// TwinCAT 3 PLC project nadaCAT
// ProgramVersion: 3.1.4024.0
// libraries:
//   Tc2_MC2, * (Beckhoff Automation GmbH)
//   Tc2_MC2_Drive, * (Beckhoff Automation GmbH)
//   Tc2_Standard, * (Beckhoff Automation GmbH)
//   Tc2_System, * (Beckhoff Automation GmbH)
//   Tc2_TcpIp, * (Beckhoff Automation GmbH)
//   Tc2_Utilities, * (Beckhoff Automation GmbH)
//   Tc3_Module, * (Beckhoff Automation GmbH)
//   VisuDialogs, * (System)
//   VisuSymbols,3.5.10.0,System
// project tree:
//   DUTs/Enums/ E_CommandList.TcTLEO (not stored), E_ServoState.TcTLEO, E_TCPState.TcTLEO (not stored)
//   DUTs/Structs/ dutCommand.TcDUT, mcInterface.TcDUT (not stored), mcOutputs.TcDUT (not stored), stConfigParams.TcDUT (not stored), stServoInterface.TcDUT (not stored), stStateTransitions.TcDUT
//   / GlobalTextList.TcGTLO (not stored), PlcTask.TcTTO (not stored), Visualization Manager.TcVMO (not stored), VISU_TASK.TcTTO
//   GVLs/ gvlMotion.TcGVL, IO.TcGVL, PLCSystem.TcGVL, ServoGVLs.TcGVL
//   POUs/FBs/ FB_AutoMotionControl.TcPOU (not stored), FB_ManualMotionControl.TcPOU, fb_StateMachine.TcPOU, FB_TCPServer.TcPOU, sfc_TCPServer.TcPOU
//   POUs/ MAIN.TcPOU
//   POUs/PRGs/ Motion.TcPOU (not stored), System.TcPOU (not stored), TCPComm.TcPOU
//   VISUs/ Main.TcVIS
//   VISUs/Templates/ MotorFaceplate.TcVIS, MotorFaceplate2.TcVIS, SysPanel.TcVIS

CONFIGURATION nadaCAT
    RESOURCE PLC ON TwinCAT3
        TASK VISU_TASK(INTERVAL := T#200000us, PRIORITY := 30);
        PROGRAM VisuElems_Visu_Prg WITH VISU_TASK : VisuElems.Visu_Prg;
    END_RESOURCE
END_CONFIGURATION

// ---- DUTs/Enums/E_ServoState.TcTLEO
{attribute 'qualified_only'}
{attribute 'strict'}
TYPE E_ServoState :
(
	DEFAULT	  := -1,
	OFF		  := 0,
	DISABLED,
	FAULTED,
	ENABLED,
	STANDBY,
	HOMING,
	MOVE_ABS,
	MOVE_REL,
	MOVE_SCAN,
	INTERLOCK_MOTION
);
END_TYPE
//  DEFAULT = '-1'

// ---- DUTs/Structs/dutCommand.TcDUT
TYPE dutCommand :
STRUCT
	eCommand 	: E_CommandList;
	arrParam	: ARRAY [1..5] OF LINT;
END_STRUCT
END_TYPE

// ---- DUTs/Structs/stStateTransitions.TcDUT
TYPE stStateTransitions :
STRUCT
	Init			: BOOL := FALSE;
	Standby			: BOOL := FALSE;
	cmdReceived		: BOOL := FALSE;
	cmdHome			: BOOL := FALSE;
	cmdScan			: BOOL := FALSE;
	cmdMTP			: BOOL := FALSE;
	cmdMovr			: BOOL := FALSE;
	cmdMova			: BOOL := FALSE;
	cmdStat			: BOOL := FALSE;
	cmdCal			: BOOL := FALSE;
	cmdParam		: BOOL := FALSE;
	cmdHomeDone		: BOOL := FALSE;
	cmdScanDone		: BOOL := FALSE;
	cmdMTPDone		: BOOL := FALSE;
	cmdMovrDone		: BOOL := FALSE;
	cmdMovaDone		: BOOL := FALSE;
	cmdStatDone		: BOOL := FALSE;
	cmdCalDone		: BOOL := FALSE;
	cmdParamDone	: BOOL := FALSE;
	cmdComplete		: BOOL := FALSE;
END_STRUCT
END_TYPE

// ---- GVLs/gvlMotion.TcGVL
{attribute 'qualified_only'}
VAR_GLOBAL
// Manual Control
servo1			: FB_ManualMotionControl;
bank1			: FB_AutoMotionControl;
manualMode 		: BOOL := TRUE;
autoMode		: BOOL;
// Server Control
cmdData 		: dutCommand;
bEnableDrive	: BOOL := FALSE;
bStartDrive		: BOOL := FALSE;
bTriggerDefault : BOOL := FALSE;
bInterlockOK	: BOOL := TRUE;
mcBankAxis		: stServoInterface;
driveStatus 	: ST_AxisStatus;	
END_VAR

// ---- GVLs/IO.TcGVL
{attribute 'qualified_only'}
VAR_GLOBAL
	/// Inputs
	bHomeSwitch 		AT %I* : BOOL;
	/// Outputs
	
END_VAR

// ---- GVLs/PLCSystem.TcGVL
{attribute 'qualified_only'}
VAR_GLOBAL
	iTaskIdx 	: DINT;
	bFirstCycle : BOOL;
END_VAR

// ---- GVLs/ServoGVLs.TcGVL
{attribute 'qualified_only'}
VAR_GLOBAL
	servo1Interface		: stServoInterface;
	servo2Interface		: stServoInterface;
	
	rTorqueLimit AT %Q*		: INT;
	rTorqueAct	 AT %I*		: INT;
	
	probe1Signal AT %I*		: WORD;
	probe1NegLatch AT %I*		: WORD;
	probe1PosLatch AT %I*		: WORD;
	
	probe1Enable AT %Q*		: WORD;
	probe1Command AT %Q*		: WORD;
	
	coeRead : FB_CoERead;
	catchWord : WORD;
	toggle : BOOL;
END_VAR

// ---- POUs/FBs/FB_ManualMotionControl.TcPOU
FUNCTION_BLOCK FB_ManualMotionControl
VAR_INPUT
	
END_VAR
VAR_OUTPUT
END_VAR
VAR_IN_OUT
	stServoInterface		: stServoInterface;
END_VAR
VAR
	
	servoPower				: MC_Power;
	servoBuffer				: MC_BufferMode := MC_Aborting;
	
	servoReset				: MC_Reset;
	servoHome				: MC_Home;
	
	servoStatus				: MC_ReadStatus;
	
	servoSetPosition		: MC_SetPosition;
	
	servoJog				: MC_Jog;
	
	servoStop				: MC_Stop;
	
	servoMoveAbsolute		: MC_MoveAbsolute;
	
	servoMoveRelative		: MC_MoveRelative;
	
	servoMoveVelocity		: MC_MoveVelocity;
	
	jogErrorID				: UDINT;
	
	errorStop: BOOL;
	disabled: BOOL;
	stopping: BOOL;
	discreteMotion: BOOL;
	continuousMotion: BOOL;
	syncMotion: BOOL;
	homing: BOOL;
	constVelocity: BOOL;
	accel: BOOL;
	decel: BOOL;
	status: ST_AxisStatus;
	
	powerInterface 		: mcInterface;
	resetInterface		: mcInterface;
	homeInterface		: mcInterface;
	jogInterface		: mcInterface;
	stopInterface		: mcInterface;
	moveAbsInterface	: mcInterface;
	moveRelInterface	: mcInterface;
	moveVelInterface	: mcInterface;
	statusInterface		: mcInterface;
	
	// State Machine Variables
	startCycle			: BOOL;
	continueToTop		: BOOL;
	continueToBottom	: BOOL;
	endAtTop			: BOOL;
	endAtBottom			: BOOL;
	moveBottomTrig			: BOOL;
	moveTopTrig				: BOOL;
	
	demoState			: fb_StateMachine;
	demoModePermissive	: BOOL;
	demoModeRun			: BOOL;
	bottomComplete		: BOOL;
	topComplete			: BOOL;
	
	servoMoveBottom		: MC_MoveAbsolute;
	servoMoveTop		: MC_MoveAbsolute;
	servoEstop			: MC_Halt;
	
	demoModePermissivesdf: INT;
END_VAR

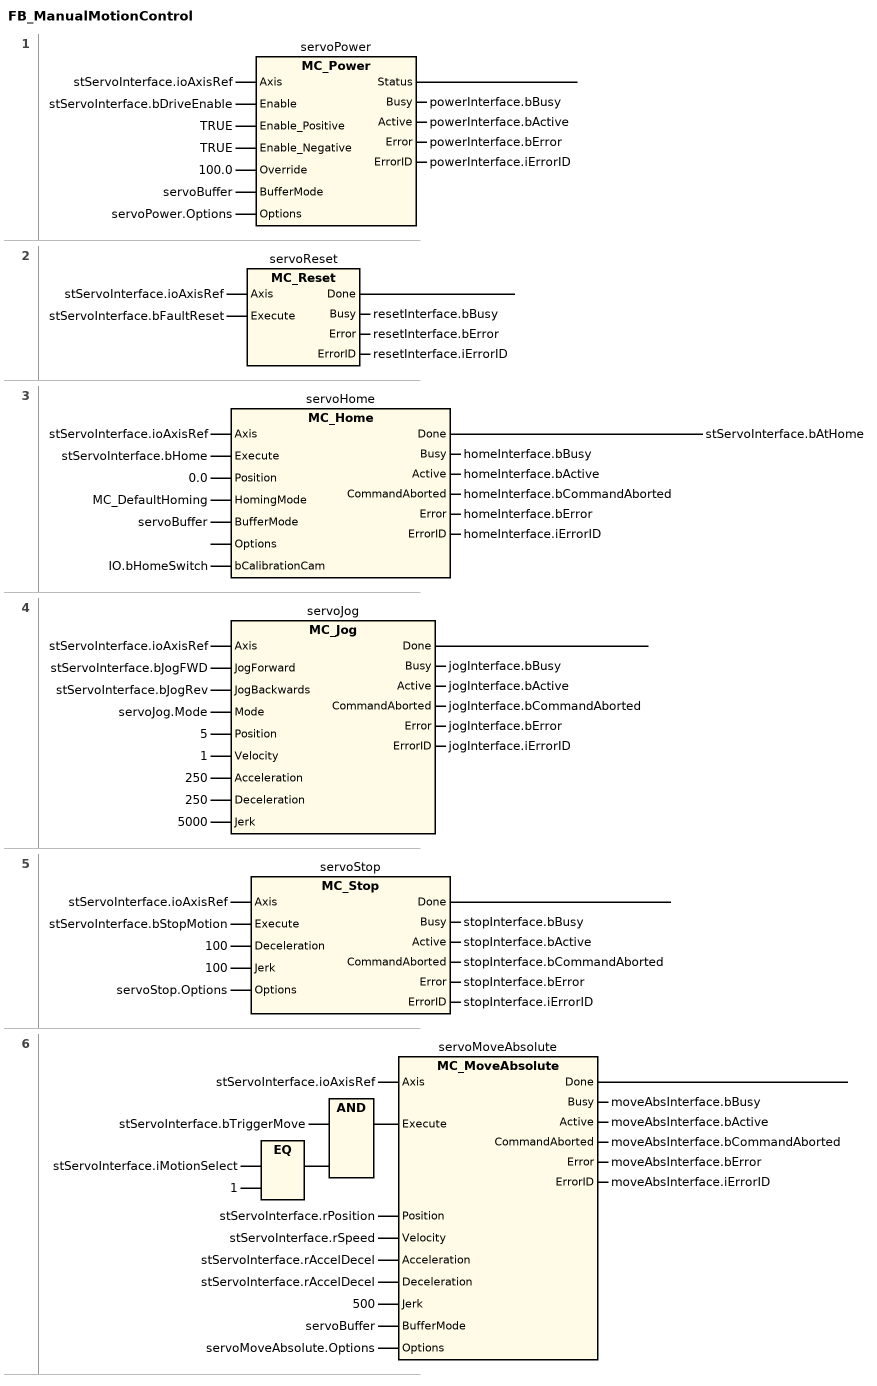
// NETWORK 1
servoPower(
    Axis := stServoInterface.ioAxisRef,
    Enable := stServoInterface.bDriveEnable,
    Enable_Positive := TRUE,
    Enable_Negative := TRUE,
    Override := 100.0,
    BufferMode := servoBuffer,
    Options := servoPower.Options,
    Busy => powerInterface.bBusy,
    Active => powerInterface.bActive,
    Error => powerInterface.bError,
    ErrorID => powerInterface.iErrorID); // MC_Power

// NETWORK 2
servoReset(
    Axis := stServoInterface.ioAxisRef,
    Execute := stServoInterface.bFaultReset,
    Busy => resetInterface.bBusy,
    Error => resetInterface.bError,
    ErrorID => resetInterface.iErrorID); // MC_Reset

// NETWORK 3
servoHome(
    Axis := stServoInterface.ioAxisRef,
    Execute := stServoInterface.bHome,
    Position := 0.0,
    HomingMode := MC_DefaultHoming,
    BufferMode := servoBuffer,
    bCalibrationCam := IO.bHomeSwitch,
    Busy => homeInterface.bBusy,
    Active => homeInterface.bActive,
    CommandAborted => homeInterface.bCommandAborted,
    Error => homeInterface.bError,
    ErrorID => homeInterface.iErrorID); // MC_Home
stServoInterface.bAtHome := servoHome.Done;

// NETWORK 4
servoJog(
    Axis := stServoInterface.ioAxisRef,
    JogForward := stServoInterface.bJogFWD,
    JogBackwards := stServoInterface.bJogRev,
    Mode := servoJog.Mode,
    Position := 5,
    Velocity := 1,
    Acceleration := 250,
    Deceleration := 250,
    Jerk := 5000,
    Busy => jogInterface.bBusy,
    Active => jogInterface.bActive,
    CommandAborted => jogInterface.bCommandAborted,
    Error => jogInterface.bError,
    ErrorID => jogInterface.iErrorID); // MC_Jog

// NETWORK 5
servoStop(
    Axis := stServoInterface.ioAxisRef,
    Execute := stServoInterface.bStopMotion,
    Deceleration := 100,
    Jerk := 100,
    Options := servoStop.Options,
    Busy => stopInterface.bBusy,
    Active => stopInterface.bActive,
    CommandAborted => stopInterface.bCommandAborted,
    Error => stopInterface.bError,
    ErrorID => stopInterface.iErrorID); // MC_Stop

// NETWORK 6
servoMoveAbsolute(
    Axis := stServoInterface.ioAxisRef,
    Execute := stServoInterface.bTriggerMove AND stServoInterface.iMotionSelect = 1,
    Position := stServoInterface.rPosition,
    Velocity := stServoInterface.rSpeed,
    Acceleration := stServoInterface.rAccelDecel,
    Deceleration := stServoInterface.rAccelDecel,
    Jerk := 500,
    BufferMode := servoBuffer,
    Options := servoMoveAbsolute.Options,
    Busy => moveAbsInterface.bBusy,
    Active => moveAbsInterface.bActive,
    CommandAborted => moveAbsInterface.bCommandAborted,
    Error => moveAbsInterface.bError,
    ErrorID => moveAbsInterface.iErrorID); // MC_MoveAbsolute

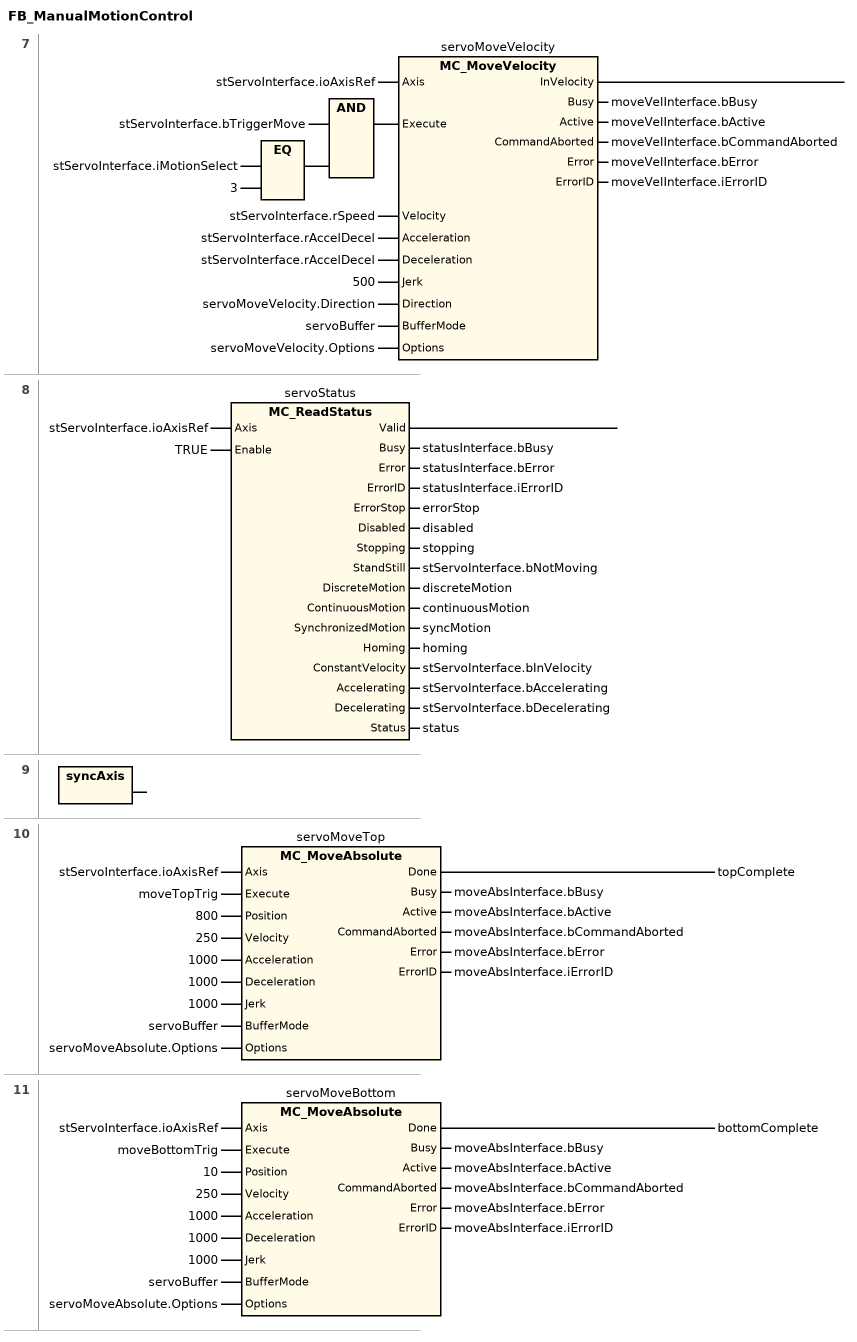
// NETWORK 7
servoMoveVelocity(
    Axis := stServoInterface.ioAxisRef,
    Execute := stServoInterface.bTriggerMove AND stServoInterface.iMotionSelect = 3,
    Velocity := stServoInterface.rSpeed,
    Acceleration := stServoInterface.rAccelDecel,
    Deceleration := stServoInterface.rAccelDecel,
    Jerk := 500,
    Direction := servoMoveVelocity.Direction,
    BufferMode := servoBuffer,
    Options := servoMoveVelocity.Options,
    Busy => moveVelInterface.bBusy,
    Active => moveVelInterface.bActive,
    CommandAborted => moveVelInterface.bCommandAborted,
    Error => moveVelInterface.bError,
    ErrorID => moveVelInterface.iErrorID); // MC_MoveVelocity

// NETWORK 8
servoStatus(
    Axis := stServoInterface.ioAxisRef,
    Enable := TRUE,
    Busy => statusInterface.bBusy,
    Error => statusInterface.bError,
    ErrorID => statusInterface.iErrorID,
    ErrorStop => errorStop,
    Disabled => disabled,
    Stopping => stopping,
    StandStill => stServoInterface.bNotMoving,
    DiscreteMotion => discreteMotion,
    ContinuousMotion => continuousMotion,
    SynchronizedMotion => syncMotion,
    Homing => homing,
    ConstantVelocity => stServoInterface.bInVelocity,
    Accelerating => stServoInterface.bAccelerating,
    Decelerating => stServoInterface.bDecelerating,
    Status => status); // MC_ReadStatus

// NETWORK 9
syncAxis();

// NETWORK 10
servoMoveTop(
    Axis := stServoInterface.ioAxisRef,
    Execute := moveTopTrig,
    Position := 800,
    Velocity := 250,
    Acceleration := 1000,
    Deceleration := 1000,
    Jerk := 1000,
    BufferMode := servoBuffer,
    Options := servoMoveAbsolute.Options,
    Busy => moveAbsInterface.bBusy,
    Active => moveAbsInterface.bActive,
    CommandAborted => moveAbsInterface.bCommandAborted,
    Error => moveAbsInterface.bError,
    ErrorID => moveAbsInterface.iErrorID); // MC_MoveAbsolute
topComplete := servoMoveTop.Done;

// NETWORK 11
servoMoveBottom(
    Axis := stServoInterface.ioAxisRef,
    Execute := moveBottomTrig,
    Position := 10,
    Velocity := 250,
    Acceleration := 1000,
    Deceleration := 1000,
    Jerk := 1000,
    BufferMode := servoBuffer,
    Options := servoMoveAbsolute.Options,
    Busy => moveAbsInterface.bBusy,
    Active => moveAbsInterface.bActive,
    CommandAborted => moveAbsInterface.bCommandAborted,
    Error => moveAbsInterface.bError,
    ErrorID => moveAbsInterface.iErrorID); // MC_MoveAbsolute
bottomComplete := servoMoveBottom.Done;

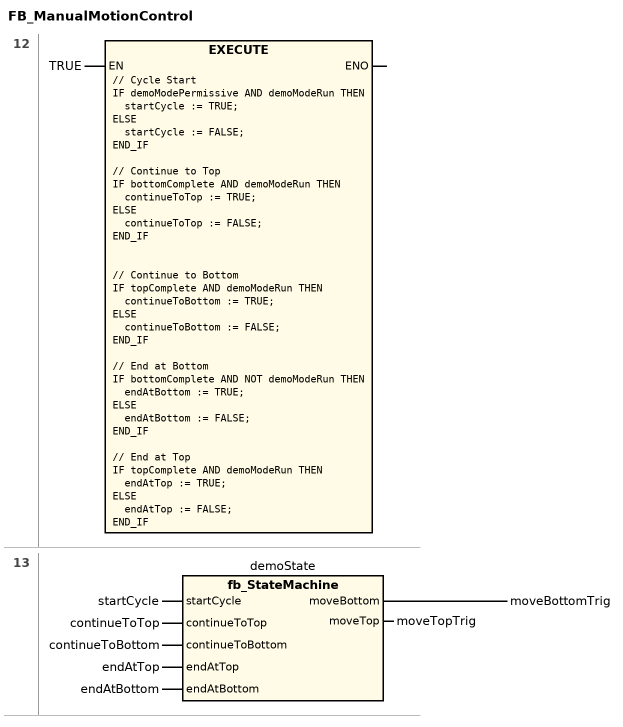
// NETWORK 12
// Cycle Start
IF demoModePermissive AND demoModeRun THEN
	startCycle := TRUE;
ELSE 
	startCycle := FALSE;
END_IF

// Continue to Top
IF bottomComplete AND demoModeRun THEN
	continueToTop := TRUE;
ELSE
	continueToTop := FALSE;
END_IF


// Continue to Bottom
IF topComplete AND demoModeRun THEN
	continueToBottom := TRUE;
ELSE
	continueToBottom := FALSE;
END_IF

// End at Bottom
IF bottomComplete AND NOT demoModeRun THEN
	endAtBottom := TRUE;
ELSE
	endAtBottom := FALSE;
END_IF

// End at Top
IF topComplete AND demoModeRun THEN
	endAtTop := TRUE;
ELSE
	endAtTop := FALSE;
END_IF

// NETWORK 13
demoState(
    startCycle := startCycle,
    continueToTop := continueToTop,
    continueToBottom := continueToBottom,
    endAtTop := endAtTop,
    endAtBottom := endAtBottom,
    moveTop => moveTopTrig); // fb_StateMachine
moveBottomTrig := demoState.moveBottom;

ACTION moveBottom:
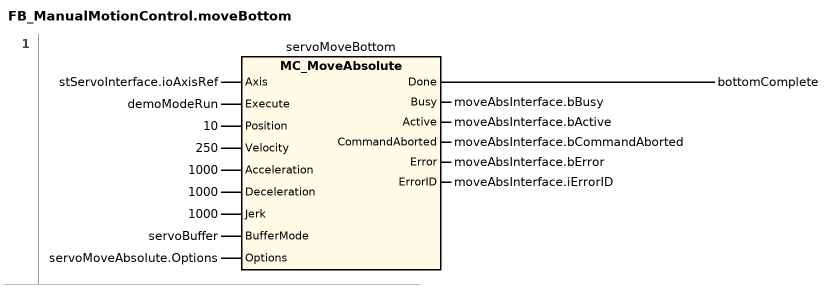
// NETWORK 1
servoMoveBottom(
    Axis := stServoInterface.ioAxisRef,
    Execute := demoModeRun,
    Position := 10,
    Velocity := 250,
    Acceleration := 1000,
    Deceleration := 1000,
    Jerk := 1000,
    BufferMode := servoBuffer,
    Options := servoMoveAbsolute.Options,
    Busy => moveAbsInterface.bBusy,
    Active => moveAbsInterface.bActive,
    CommandAborted => moveAbsInterface.bCommandAborted,
    Error => moveAbsInterface.bError,
    ErrorID => moveAbsInterface.iErrorID); // MC_MoveAbsolute
bottomComplete := servoMoveBottom.Done;
END_ACTION

ACTION moveTop:
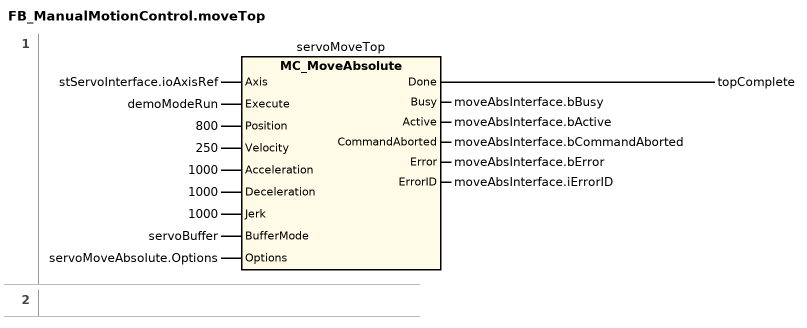
// NETWORK 1
servoMoveTop(
    Axis := stServoInterface.ioAxisRef,
    Execute := demoModeRun,
    Position := 800,
    Velocity := 250,
    Acceleration := 1000,
    Deceleration := 1000,
    Jerk := 1000,
    BufferMode := servoBuffer,
    Options := servoMoveAbsolute.Options,
    Busy => moveAbsInterface.bBusy,
    Active => moveAbsInterface.bActive,
    CommandAborted => moveAbsInterface.bCommandAborted,
    Error => moveAbsInterface.bError,
    ErrorID => moveAbsInterface.iErrorID); // MC_MoveAbsolute
topComplete := servoMoveTop.Done;

// NETWORK 2
END_ACTION

ACTION syncAxis:
CASE stServoInterface.ioAxisRef.NcToPlc.AxisState OF
	0 : // Inactive
	
	1 : // Running
		
	3 : // Phase_VeloConst
		stServoInterface.bInVelocity := TRUE;
	4 : // Phase_AccPos
		stServoInterface.bAccelerating := TRUE;
	5 : // Phase_AccNeg
		stServoInterface.bDecelerating := TRUE;
END_CASE

// Feedback

stServoInterface.rActualPosition := stServoInterface.ioAxisRef.NcToPlc.ActPos;

stServoInterface.rActualSpeed := stServoInterface.ioAxisRef.NcToPlc.ActVelo;

// Motion Status
stServoInterface.bDriveEnabled:= NOT(disabled);
stServoInterface.bMoving := NOT(stServoInterface.bNotMoving AND disabled);
stServoInterface.bFaulted := statusInterface.bError;

// Drive Control

// Demo Mode
IF stServoInterface.iMotionSelect = 1 THEN
	demoModePermissive := TRUE;
ELSE
	demoModePermissive := FALSE;
END_IF

IF demoModePermissive AND (stServoInterface.bDemoModeStart OR demoModeRun) AND NOT stServoInterface.bDemoModeStop THEN
	demoModeRun := TRUE;
ELSE
	demoModeRun := FALSE;
END_IF
END_ACTION

END_FUNCTION_BLOCK

// ---- POUs/FBs/fb_StateMachine.TcPOU
FUNCTION_BLOCK fb_StateMachine
VAR_INPUT
	startCycle 			: BOOL;
	continueToTop		: BOOL;
	continueToBottom	: BOOL;
	endAtTop			: BOOL;
	endAtBottom			: BOOL;
END_VAR
VAR_OUTPUT
	moveBottom			: BOOL;
	moveTop				: BOOL;
END_VAR
VAR
END_VAR

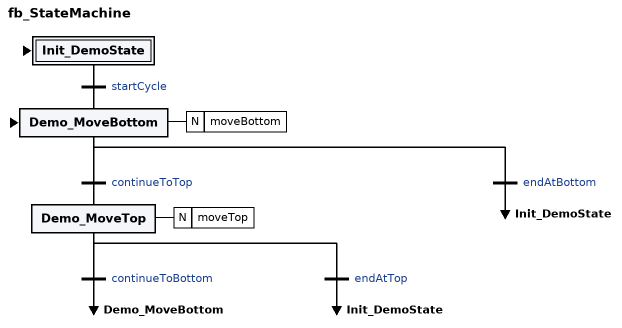
INITIAL_STEP Init_DemoState:
END_STEP
TRANSITION FROM Init_DemoState TO Demo_MoveBottom
    := startCycle;
END_TRANSITION
STEP Demo_MoveBottom:
    moveBottom(N);
END_STEP
TRANSITION FROM Demo_MoveBottom TO Demo_MoveTop
    := continueToTop;
END_TRANSITION
TRANSITION FROM Demo_MoveBottom TO Init_DemoState
    := endAtBottom;
END_TRANSITION
STEP Demo_MoveTop:
    moveTop(N);
END_STEP
TRANSITION FROM Demo_MoveTop TO Demo_MoveBottom
    := continueToBottom;
END_TRANSITION
TRANSITION FROM Demo_MoveTop TO Init_DemoState
    := endAtTop;
END_TRANSITION
// branch label Branch0_DemoState

END_FUNCTION_BLOCK

// ---- POUs/FBs/FB_TCPServer.TcPOU
FUNCTION_BLOCK FB_TCPServer
VAR_INPUT
    sLocalHost: T_IPv4Addr;
    nLocalPort: UDINT;
    bStartCommunication : BOOL;
END_VAR
VAR_OUTPUT
    bConnected: BOOL;
    cmdData : dutCommand;  // Command data structure including eCommand and arrParam
    bBusy: BOOL;
    bError: BOOL;
    nErrorID: UDINT;
    sSendData: STRING(255);  // Define this output if it represents data being sent
END_VAR
VAR
    bAccepted: BOOL;
	bReturn: BOOL;  // Define bReturn for _SendServerResponse calls
    bHasParam: BOOL;
    iState: INT;
	ii	  : INT;
    hListener: T_HSOCKET;
    hSocket: T_HSOCKET;
    fbSocketAccept: FB_SocketAccept;
    fbSocketListen: FB_SocketListen;
    fbSocketReceive: FB_SocketReceive;
    fbSocketClose: FB_SocketClose;
	fbSocketCloseAll: FB_SocketCloseAll;
    fbSocketSend: FB_SocketSend;
    sReadData: STRING(255);
    nLength: INT;
    sCommand: STRING(255);
    sParam: STRING(255);
END_VAR

ServerConnection();
IF bConnected THEN
	ServerApplication();
END_IF

METHOD _ParseCommand : E_CommandList
VAR
    nParamStart : INT;
    nSpacePos : INT;
    nTempParam : LINT;
    sBuff : STRING(255);  // Buffer for the main parsing steps
    sTail : STRING := '$0D$0A';  // Tail for CR LF removal
END_VAR
// Initialize outputs
FOR ii := 1 TO 5 DO
	cmdData.arrParam[ii] := 0;  // Reset parameter array
END_FOR
bHasParam := FALSE;

// Step 1: Prepare command buffer (sBuff) by removing trailing CR LF
nLength := LEN(sReadData);
IF nLength > 2 THEN
    sBuff := LEFT(sReadData, nLength - 2);  // Remove CR LF
ELSE
    sBuff := sReadData;  // Use original if no CR LF found
END_IF

// Step 2: Find the first space in sBuff to separate the command from parameters
nSpacePos := FIND(sBuff, ' ');
IF nSpacePos > 0 THEN
    // Split command and parameter parts
    sCommand := LEFT(sBuff, nSpacePos - 1);
    nParamStart := nSpacePos + 1;
    sParam := MID(sBuff, LEN(sBuff) - nParamStart + 1, nParamStart);
    
	// Split sParam by commas
    nLength := LEN(sParam);
    IF nLength > 0 THEN
        ii := 1;
        WHILE (ii <= 5) AND (nLength > 0) DO
            nSpacePos := FIND(sParam, ',');
            IF nSpacePos > 0 THEN
                sBuff := LEFT(sParam, nSpacePos - 1);
                sParam := MID(sParam, nLength - nSpacePos, nSpacePos + 1);
                nLength := LEN(sParam);
            ELSE
                sBuff := sParam;
                nLength := 0;
            END_IF
            nTempParam := STRING_TO_LINT(sBuff);
            IF nTempParam <> 0 THEN
                cmdData.arrParam[ii] := nTempParam;  // Store parameter
                bHasParam := TRUE;
            END_IF
            ii := ii + 1;
        END_WHILE
    END_IF
ELSE
    // If no space is found, assume the whole sBuff is the command
    sCommand := sBuff;
    sParam := '';
END_IF

// Step 3: Command matching and parameter handling
IF sCommand = 'LIST' THEN
    _ParseCommand := E_CommandList.LIST;

ELSIF sCommand = 'HOM' THEN
    _ParseCommand := E_CommandList.HOM;

ELSIF sCommand = 'SCAN' THEN
    _ParseCommand := E_CommandList.SCAN;
	IF sParam <> '' THEN
		bHasParam := TRUE;
	END_IF

ELSIF sCommand = 'MTP' THEN
    _ParseCommand := E_CommandList.MTP;

ELSIF sCommand = 'MOVR' THEN
    _ParseCommand := E_CommandList.MOVR;
    IF sParam <> '' THEN
        nTempParam := STRING_TO_LINT(sParam);
        IF nTempParam <> 0 THEN
            cmdData.arrParam[1] := nTempParam;  // Store MOVR parameter
            bHasParam := TRUE;
        END_IF
    END_IF

ELSIF sCommand = 'MOVA' THEN
    _ParseCommand := E_CommandList.MOVA;
    IF sParam <> '' THEN
        nTempParam := STRING_TO_LINT(sParam);
        IF nTempParam <> 0 THEN
            cmdData.arrParam[1] := nTempParam;  // Store MOVA parameter
            bHasParam := TRUE;
        END_IF
    END_IF

ELSIF sCommand = 'STAT' THEN
    _ParseCommand := E_CommandList.STAT;

ELSIF sCommand = 'CALIB' THEN
    _ParseCommand := E_CommandList.CALIB;

ELSIF sCommand = 'PARAM' THEN
    _ParseCommand := E_CommandList.PARAM;

ELSE
    _ParseCommand := E_CommandList.ERR;  // Unknown command
END_IF
END_METHOD

METHOD _SendServerResponse : BOOL
VAR_INPUT
	sResponseText : STRING(255);
END_VAR
VAR
    sCRLF : STRING := '$0D$0A';
    sFinalResponse : STRING(255);
    nResponseSize : INT;
END_VAR
// Build the full response
sFinalResponse := CONCAT(sResponseText, sCRLF);

// Copy response to send buffer
nResponseSize := LEN(sFinalResponse);
memcpy(ADR(sSendData), ADR(sFinalResponse), nResponseSize);

// Null-terminate
sSendData[nResponseSize] := 0;
END_METHOD

METHOD MotionConnection : BOOL
VAR_INPUT
END_VAR
END_METHOD

METHOD ServerApplication : BOOL
VAR
    eCommandTemp: E_CommandList;
	sResponseBuff : STRING(255);
END_VAR
CASE iState OF
    30: // Receive Data
        fbSocketReceive(
            sSrvNetId := '',
            hSocket := hSocket,
            cbLen := SIZEOF(sReadData),
            pDest := ADR(sReadData),
            bExecute := TRUE,
            tTimeout := T#4S,
            bBusy => ,
            bError => bError,
            nErrId => nErrorID
        );

        IF NOT fbSocketReceive.bBusy THEN
            fbSocketReceive(bExecute := FALSE);
            IF fbSocketReceive.nRecBytes <> 0 THEN
                fbSocketSend(bExecute := FALSE);
                iState := 300;
            END_IF
        END_IF

        // Close connection when error occurs or trigger is set
        IF fbSocketReceive.bError OR (NOT bStartCommunication) THEN
            iState := iState + 10;
        END_IF

    300: // Parse Data
        eCommandTemp := _ParseCommand();
        cmdData.eCommand := eCommandTemp;  // Set parsed command to cmdData

        CASE cmdData.eCommand OF
            E_CommandList.LIST:
                bReturn := _SendServerResponse('LIST, HOM, SCAN, MTP, MOVR, MOVA, STAT, CALIB, PARAM');
            
            E_CommandList.HOM:
                bReturn := _SendServerResponse('HOM');

            E_CommandList.SCAN:
				sResponseBuff := 'SCAN ';
				IF bHasParam THEN
					FOR ii := 1 TO 5 DO
						cmdData.arrParam[ii] := cmdData.arrParam[ii];
						IF cmdData.arrParam[ii] <> 0 THEN
							sResponseBuff := CONCAT(sResponseBuff,LINT_TO_STRING(cmdData.arrParam[ii]));
							sResponseBuff := CONCAT(sResponseBuff, ' ');
						END_IF
					END_FOR
				END_IF
                bReturn := _SendServerResponse(sResponseBuff);

            E_CommandList.MTP:
                bReturn := _SendServerResponse('MTP');

            E_CommandList.MOVR:
                IF bHasParam THEN
                    cmdData.arrParam[1] := cmdData.arrParam[1];  // Use arrParam[1] for MOVA
                END_IF
				bReturn := _SendServerResponse('MOVR');

            E_CommandList.MOVA:
                IF bHasParam THEN
                    cmdData.arrParam[1] := cmdData.arrParam[1];  // Use arrParam[1] for MOVA
                END_IF
                bReturn := _SendServerResponse('MOVA');

            E_CommandList.STAT:
                bReturn := _SendServerResponse('STAT');

            E_CommandList.CALIB:
                bReturn := _SendServerResponse('CALIB');

            E_CommandList.PARAM:
                bReturn := _SendServerResponse('PARAM');

            E_CommandList.ERR:
                bReturn := _SendServerResponse('ERR');
        END_CASE
        iState := 34;

    34: // Clear ReceiveBuffer after processing
        memset(ADR(sReadData), 0, SIZEOF(sReadData));
        iState := 35;

    35: // Send Data
        fbSocketSend(
            sSrvNetId := '',
            hSocket := hSocket,
            cbLen := SIZEOF(sSendData),
            pSrc := ADR(sSendData),
            bExecute := TRUE,
            tTimeout := T#3S,
            bBusy => ,
            bError => bError,
            nErrId => nErrorID
        );

        IF NOT fbSocketSend.bBusy THEN
            memset(ADR(sSendData), 0, SIZEOF(sSendData));
            cmdData.eCommand := E_CommandList.NULL;
            iState := iState - 5;
        ELSIF fbSocketSend.bError THEN
            iState := iState + 5;
        END_IF
END_CASE
END_METHOD

METHOD ServerConnection : BOOL
VAR
END_VAR
CASE iState OF
0: // Init State
    IF bStartCommunication = TRUE THEN
        fbSocketListen(bExecute := FALSE);
        fbSocketAccept(bExecute := FALSE);
        fbSocketCloseAll(bExecute := FALSE);
        fbSocketClose(bExecute:= FALSE);
		bConnected := FALSE;
        bBusy := TRUE;
        iState := iState + 10;
    ELSE
        bBusy := FALSE;
    END_IF

10: // Open Listener-Socket
    fbSocketListen(
        sSrvNetId:= '',                                                 // Local NetID
        sLocalHost:= sLocalHost,                                         // Local IP
        nLocalPort:= nLocalPort,                                         // Local Port
        bExecute:= TRUE, 
        tTimeout:= T#4S, 
        bBusy=> , 
        bError=> bError, 
        nErrId=> nErrorID,
        hListener=> hListener);                                          // Handle of Listener Socket

    IF hListener.handle <> 0 THEN
        iState := iState + 10;    
    ELSIF bError THEN
        iState := 40; // Error state
    END_IF

20: // Accept Client Connection
    fbSocketAccept(
        sSrvNetId:= '',         
        hListener:= hListener,                                           // Handle of Listener Socket
        bExecute:= TRUE, 
        tTimeout:= T#4S, 
        bAccepted=> bAccepted, 
        bBusy=> , 
        bError=> bError, 
        nErrId=> nErrorID,
        hSocket=> hSocket);                                              // Connection Handle

    IF NOT fbSocketAccept.bBusy THEN
        fbSocketAccept(bExecute := FALSE);
    END_IF
				   
    IF bError THEN
        iState := 40;  // Error state
	ELSIF hSocket.handle <> 0 THEN
        bConnected := TRUE;
		iState := iState + 10;											// Step into ServerApplication
	END_IF

40: // Error Handling    
    fbSocketClose(                                                        // Close Listener-Socket
        sSrvNetId:= '', 
        hSocket:= hListener, 
        bExecute:= TRUE, 
        tTimeout:= T#4S, 
        bBusy=> , 
        bError=> bError, 
        nErrId=> nErrorID);        

    IF (NOT fbSocketClose.bBusy) OR fbSocketClose.bError THEN
        hListener.handle := 0;
        iState := iState + 1;
    END_IF

41:    
    fbSocketClose(bExecute := FALSE);
    iState := iState + 1;

42: // Close Connection Socket
    fbSocketClose(
        sSrvNetId:= '', 
        hSocket:= hSocket, 
        bExecute:= TRUE, 
        tTimeout:= T#4S, 
        bBusy=> , 
        bError=> bError, 
        nErrId=> nErrorID);

    IF NOT (fbSocketClose.bBusy) OR fbSocketClose.bError THEN
        hSocket.handle := 0;    
        iState := 0;
        bConnected := FALSE;
    END_IF
END_CASE
END_METHOD

END_FUNCTION_BLOCK

// ---- POUs/FBs/sfc_TCPServer.TcPOU
FUNCTION_BLOCK sfc_TCPServer
VAR_INPUT
	sLocalHost: T_IPv4Addr;
	nLocalPort: UDINT;
	bStartCommunication : BOOL;
END_VAR
VAR_OUTPUT
	bConnected: BOOL;
	eCommand : E_CommandList;
	sSendData: STRING(255);
	bBusy: BOOL;	
	bError: BOOL;
	nErrorID: UDINT;
END_VAR
VAR
	
	// State Vars
	iState				: INT;
	xInit				: R_TRIG;
	xOpenSocket			: R_TRIG;
	xError0				: R_TRIG;
	xError1				: R_TRIG;
	xError2				: R_TRIG;
	xError3				: R_TRIG;
	xError4				: R_TRIG;
	xError5				: R_TRIG;
	xAcceptConnection	: R_TRIG;
	xReceiveData		: R_TRIG;
	xParseData			: R_TRIG;
	xClearBuff			: R_TRIG;
	xSendData			: R_TRIG;
	xErrHandle			: R_TRIG;
	xPreClose			: R_TRIG;
	xCloseSocket		: R_TRIG;
	xReset				: R_TRIG;
	
	hListener: T_HSOCKET;
	hSocket: T_HSOCKET;
	fbSocketAccept: FB_SocketAccept;
	fbSocketListen: FB_SocketListen;
	fbLinkStatus: FB_IpAdapterGetLinkStatus;
	fbSocketReceive: FB_SocketReceive;
	fbSocketClose: FB_SocketClose;
	fbSocketCloseAll: FB_SocketCloseAll;
	fbSocketSend: FB_SocketSend;
	bAcceptExecute: BOOL;
	bAccepted: BOOL;
	bLinkError: BOOL;
	bStatusExecute: BOOL;
	
	ReceiveCounter: UDINT;
	sReadData: STRING(255);
	
	bSendTrigger: BOOL;
	
	// String Parse
    nLength : INT;
	sCommand : STRING(255);
	sTail	 : STRING(255);
	sBuff    : STRING(255);
	// Server Response
	bReturn : BOOL;
END_VAR

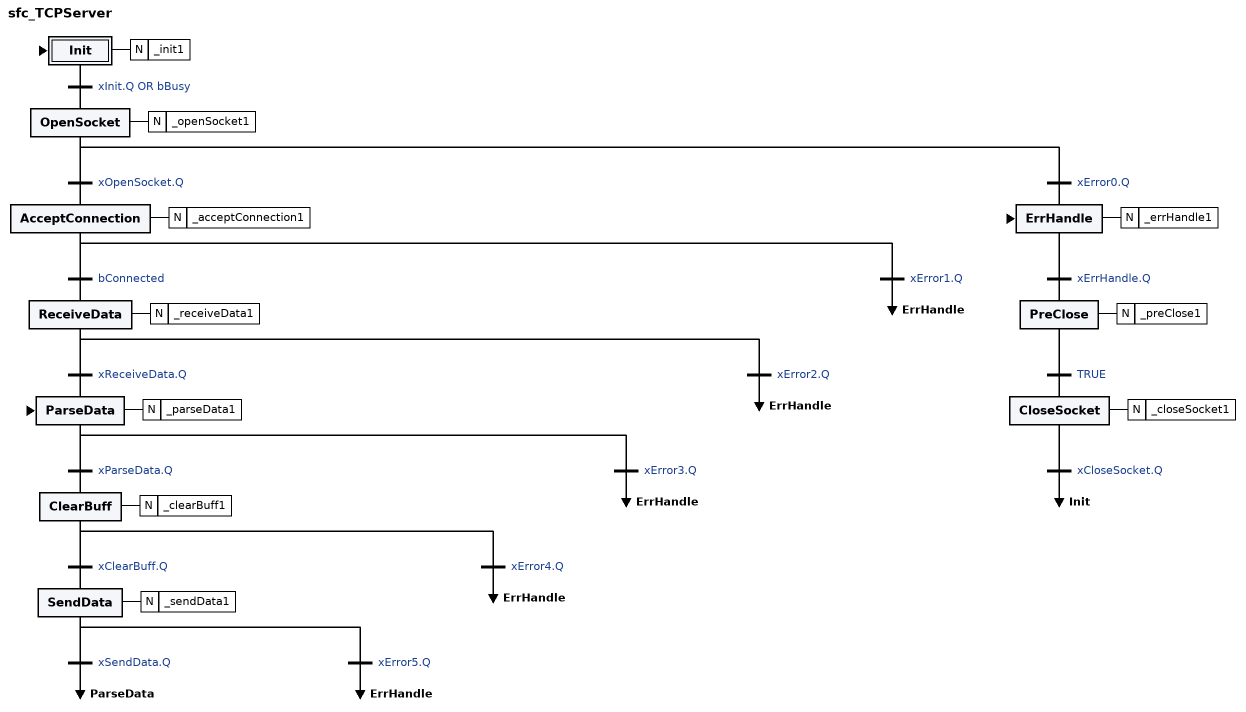
INITIAL_STEP Init:
    _init1(N);
END_STEP
TRANSITION FROM Init TO OpenSocket
    := xInit.Q OR bBusy;
END_TRANSITION
STEP OpenSocket:
    _openSocket1(N);
END_STEP
TRANSITION FROM OpenSocket TO AcceptConnection
    := xOpenSocket.Q;
END_TRANSITION
TRANSITION FROM OpenSocket TO ErrHandle
    := xError0.Q;
END_TRANSITION
STEP ErrHandle:
    _errHandle1(N);
END_STEP
TRANSITION FROM ErrHandle TO PreClose
    := xErrHandle.Q;
END_TRANSITION
STEP PreClose:
    _preClose1(N);
END_STEP
TRANSITION FROM PreClose TO CloseSocket
    := TRUE;
END_TRANSITION
STEP CloseSocket:
    _closeSocket1(N);
END_STEP
TRANSITION FROM CloseSocket TO Init
    := xCloseSocket.Q;
END_TRANSITION
STEP AcceptConnection:
    _acceptConnection1(N);
END_STEP
TRANSITION FROM AcceptConnection TO ReceiveData
    := bConnected;
END_TRANSITION
TRANSITION FROM AcceptConnection TO ErrHandle
    := xError1.Q;
END_TRANSITION
STEP ReceiveData:
    _receiveData1(N);
END_STEP
TRANSITION FROM ReceiveData TO ParseData
    := xReceiveData.Q;
END_TRANSITION
TRANSITION FROM ReceiveData TO ErrHandle
    := xError2.Q;
END_TRANSITION
STEP ParseData:
    _parseData1(N);
END_STEP
TRANSITION FROM ParseData TO ClearBuff
    := xParseData.Q;
END_TRANSITION
TRANSITION FROM ParseData TO ErrHandle
    := xError3.Q;
END_TRANSITION
STEP ClearBuff:
    _clearBuff1(N);
END_STEP
TRANSITION FROM ClearBuff TO SendData
    := xClearBuff.Q;
END_TRANSITION
TRANSITION FROM ClearBuff TO ErrHandle
    := xError4.Q;
END_TRANSITION
STEP SendData:
    _sendData1(N);
END_STEP
TRANSITION FROM SendData TO ParseData
    := xSendData.Q;
END_TRANSITION
TRANSITION FROM SendData TO ErrHandle
    := xError5.Q;
END_TRANSITION

ACTION _acceptConnection1:
fbSocketAccept(
	sSrvNetId:= '',         
	hListener:= hListener,                                           // Handle of Listener Socket
	bExecute:= TRUE, 
	tTimeout:= T#4S, 
	bAccepted=> bAccepted, 
	bBusy=> , 
	bError=> bError, 
	nErrId=> nErrorID,
	hSocket=> hSocket);                                              // Connection Handle

xAcceptConnection(CLK:=(hSocket.handle <> 0));
IF NOT fbSocketAccept.bBusy THEN
	fbSocketAccept(bExecute := FALSE);
END_IF

fbLinkStatus(sSrvNetId:= '',
				   sLocalHost := sLocalHost,
				   bExecute := bStatusExecute,
				   tTimeout := T#4S,
				   bLinkError => bLinkError);
	   

IF hSocket.handle <> 0 THEN
	bConnected := TRUE;									
END_IF
xError1(CLK:=bError);
END_ACTION

ACTION _clearBuff1:

// Clear ReceiveBuffer after processing
xClearBuff(CLK:= (memset(ADR(sReadData), 0, SIZEOF(sReadData))>0));
(*memset(ADR(sServerEcho), 0, SIZEOF(sServerEcho));
memset(ADR(sEchoFooter), 0, SIZEOF(sEchoFooter));
memset(ADR(sEchoHeader), 0, SIZEOF(sEchoHeader));*)        

{'warning': Need TO ADD conditional here}
END_ACTION

ACTION _closeSocket1:

fbSocketClose(
	sSrvNetId:= '', 
	hSocket:= hSocket, 
	bExecute:= TRUE, 
	tTimeout:= T#4S, 
	bBusy=> , 
	bError=> bError, 
	nErrId=> nErrorID);


IF NOT (fbSocketClose.bBusy) OR fbSocketClose.bError THEN
	hSocket.handle := 0;    
	bConnected := FALSE;
END_IF
xCloseSocket(CLK:=(NOT (fbSocketClose.bBusy) OR fbSocketClose.bError));
END_ACTION

ACTION _errHandle1:

// Error Handling    
fbSocketClose(                                                        // Close Listener-Socket
	sSrvNetId:= '', 
	hSocket:= hListener, 
	bExecute:= TRUE, 
	tTimeout:= T#4S, 
	bBusy=> , 
	bError=> bError, 
	nErrId=> nErrorID);        

IF (NOT fbSocketClose.bBusy) OR fbSocketClose.bError THEN
	hListener.handle := 0;
END_IF
xErrHandle(CLK:=((NOT fbSocketClose.bBusy) OR fbSocketClose.bError));
END_ACTION

ACTION _init1:
xInit(CLK:=bStartCommunication);
IF bStartCommunication = TRUE THEN
	fbSocketListen(bExecute := FALSE);
	fbSocketAccept(bExecute := FALSE);
	fbSocketCloseAll(bExecute := FALSE);
	fbSocketClose(bExecute:= FALSE);
	bConnected := FALSE;
	bBusy := TRUE;
	

ELSE
	bBusy := FALSE;
END_IF
END_ACTION

ACTION _openSocket1:

// Open Listener-Socket
fbSocketListen(
	sSrvNetId:= '',                                                 // Local NetID
	sLocalHost:= sLocalHost,                                         // Local IP
	nLocalPort:= nLocalPort,                                         // Local Port
	bExecute:= TRUE, 
	tTimeout:= T#4S, 
	bBusy=> , 
	bError=> bError, 
	nErrId=> nErrorID,
	hListener=> hListener);                                          // Handle of Listener Socket
	
xOpenSocket(CLK:=hListener.handle <> 0);
xError0(CLK:= bError);
END_ACTION

METHOD _ParseCommand : INT
VAR_INPUT
END_VAR
// Step 1: Parse out the command and tail
nLength := LEN(sReadData);
sTail := CONCAT('$0D','$0A');
IF nLength > 2 THEN
    sCommand := LEFT(sReadData, nLength - 2);  // Remove CR LF
END_IF

// Step 2: Command matching
IF sCommand = 'LIST' THEN
    _ParseCommand := E_CommandList.LIST;
ELSIF sCommand = 'HOM' THEN
    _ParseCommand := E_CommandList.HOM;
ELSIF sCommand = 'SCAN' THEN
    _ParseCommand := E_CommandList.SCAN;
ELSIF sCommand = 'MTP' THEN
    _ParseCommand := E_CommandList.MTP;
ELSIF sCommand = 'MOVR' THEN
    _ParseCommand := E_CommandList.MOVR;
ELSIF sCommand = 'MOVA' THEN
    _ParseCommand := E_CommandList.MOVA;
ELSIF sCommand = 'STAT' THEN
    _ParseCommand := E_CommandList.STAT;
ELSIF sCommand = 'CALIB' THEN
    _ParseCommand := E_CommandList.CALIB;
ELSIF sCommand = 'PARAM' THEN
    _ParseCommand := E_CommandList.PARAM;
ELSE
    _ParseCommand := E_CommandList.ERR;  // Unknown command
END_IF
END_METHOD

ACTION _parseData1:

// Parse Data
	eCommand := _ParseCommand();
	CASE eCommand OF
		E_CommandList.LIST:
			// List out available command
			bReturn := _SendServerResponse('LIST, HOM, SCAN, MTP, MOVR, MOVA, STAT, CALIB, PARAM');
		E_CommandList.HOM:
			// Home
			bReturn := _SendServerResponse('HOM');
		E_CommandList.SCAN:
			// Scan
			bReturn := _SendServerResponse('SCAN');
		E_CommandList.MTP:
			// Move to Pod
			bReturn := _SendServerResponse('MTP');
		E_CommandList.MOVR:
			// Move Relative
			bReturn := _SendServerResponse('MOVR');
		E_CommandList.MOVA:
			// Move Absolute
			bReturn := _SendServerResponse('MOVA');
		E_CommandList.STAT:
			// Machine Status
			bReturn := _SendServerResponse('STAT');
		E_CommandList.CALIB:
			// Machine Calibration Scan
			bReturn := _SendServerResponse('CALIB');
		E_CommandList.PARAM:
			// Set Parameters Mode
			bReturn := _SendServerResponse('PARAM');
		E_CommandList.ERR:
			// Command error
			bReturn := _SendServerResponse('ERR');
	END_CASE
	xParseData(CLK:= (eCommand <> E_CommandList.NULL));
	//_ParseData := TRUE;
	{'warning': Need to add conditional here to prevent race condition}
END_ACTION

ACTION _preClose1:

fbSocketClose(bExecute := FALSE);
END_ACTION

ACTION _receiveData1:

// Receive Data
fbSocketReceive(                                                     // Check cyclically for new client data 
	sSrvNetId:= '', 
	hSocket:= hSocket, 
	cbLen:= SIZEOF(sReadData), 
	pDest:= ADR(sReadData), 
	bExecute:= TRUE,                                                 
	tTimeout:= T#4S, 
	bBusy=> , 
	bError=> bError, 
	nErrId=> nErrorID,
	nRecBytes=> );

IF NOT fbSocketReceive.bBusy THEN
	fbSocketReceive(bExecute := FALSE);
	
	IF fbSocketReceive.nRecBytes <> 0 THEN                            // Switch to send-state when data are received
		fbSocketSend(bExecute := FALSE);             
		
		
	END_IF
END_IF
xReceiveData(CLK := fbSocketReceive.nRecBytes <> 0);
xError2(CLK:=(fbSocketReceive.bError OR (NOT bStartCommunication)));
// Close connection when error is occurring or trigger is set
END_ACTION

ACTION _sendData1:

// Send Data
fbSocketSend(                                                        // Send Data to client
	sSrvNetId:= '', 
	hSocket:= hSocket, 
	cbLen:= SIZEOF(sSendData), 
	pSrc:= ADR(sSendData),
	bExecute:= TRUE, 
	tTimeout:= T#3S, 
	bBusy=> , 
	bError=> bError, 
	nErrId=> nErrorID);    

IF NOT fbSocketSend.bBusy THEN                                        // Switch back to receiving state after sending
	memset(ADR(sSendData), 0, SIZEOF(sSendData));
	eCommand := E_CommandList.NULL;
END_IF
xSendData(CLK:=NOT fbSocketSend.bBusy);
xError5(CLK:=fbSocketSend.bError);
END_ACTION

METHOD _SendServerResponse : BOOL
VAR_INPUT
	sResponseText : STRING(255);
END_VAR
VAR
    sCRLF : STRING := '$0D$0A';
    sFinalResponse : STRING(255);
    nResponseSize : INT;
END_VAR
// Build the full response
sFinalResponse := CONCAT(sResponseText, sCRLF);

// Copy response to send buffer
nResponseSize := LEN(sFinalResponse);
memcpy(ADR(sSendData), ADR(sFinalResponse), nResponseSize);

// Null-terminate
sSendData[nResponseSize] := 0;
END_METHOD

METHOD transit : BOOL
VAR_INPUT
    xCondition : BOOL;  // Input condition for transition
    xReset : BOOL;      // Input to reset the condition
END_VAR
VAR_OUTPUT
    bTransitioned : BOOL;  // Output TRUE if transition occurs
END_VAR
VAR
    rTrig : R_TRIG;  // Rising edge detector
END_VAR
// Initialize default output
bTransitioned := FALSE;

// Perform rising edge detection on the input condition
rTrig(CLK := xCondition);

// If a rising edge is detected, it means a transition is triggered
IF rTrig.Q THEN
    bTransitioned := TRUE;  // Transition has occurred
END_IF

// Reset the condition if requested to close the transition
IF xReset THEN
    bTransitioned := FALSE;  // Clear transition flag
END_IF

// Return the result of the transition
transit := bTransitioned;
END_METHOD

END_FUNCTION_BLOCK

// ---- POUs/MAIN.TcPOU
PROGRAM MAIN
VAR

END_VAR

// System Control
PLCSystem.iTaskIdx  := GETCURTASKINDEXEX();
System(iTaskIdx 	:= PLCSystem.iTaskIdx,
	   bFirstCycle  := PLCSystem.bFirstCycle);

ServoGVLs.coeRead(Axis:= servoGVLs.servo1Interface.ioAxisRef,
				  Index := 16#2191,
				  SubIndex := 16#01,
				  Execute := servoGVLs.toggle,
				  Busy =>,
				  pDstBuf := ADR(servoGVLs.catchWord),
				  BufLen := SIZEOF(servoGVLs.catchWord));

// TCP Connection

TCPComm(cmdData => gvlMotion.cmdData);
// Mode Control
gvlMotion.autoMode := NOT gvlMotion.manualMode;
IF gvlMotion.manualMode THEN
	gvlMotion.servo1(stServoInterface := servoGVLs.servo1Interface);
END_IF
// Servo 1 Auto Control via Server
gvlMotion.bank1(
	   cmdData := gvlMotion.cmdData,
	   bEnableDrive := gvlMotion.bEnableDrive,
	   bStartDrive := gvlMotion.bStartDrive,
	   bInterlockOK := gvlMotion.bInterlockOK,
	   bTriggerDefault := gvlMotion.bTriggerDefault,
	   driveStatus => gvlMotion.driveStatus,
	   mcBankAxis := ServoGVLs.servo1Interface);

END_PROGRAM

// ---- POUs/PRGs/TCPComm.TcPOU
PROGRAM TCPComm
VAR_INPUT
nServer1Port				: UDINT 				:= 12000;
sServer1Host				: T_IPv4Addr 			:= '192.168.5.1';
END_VAR
VAR_OUTPUT
	cmdData			: dutCommand;
	eCommand		: E_CommandList;
	rParam			: REAL;
END_VAR
VAR
	bInit: BOOL := TRUE;
	fbSocketCloseAll: FB_SocketCloseAll; 
	bSocketCloseError: BOOL;
	nSocketCloseError: UDINT;
	
	fbTcpEchoServer1				: FB_TCPServer;
		sServerReceivedData			: STRING(255);
		bStartServer1Communication	: BOOL 					:= TRUE;
		bServer1Connected			: BOOL;
		sServerData					: STRING(255);
		bServer1Busy				: BOOL;
		bServer1Error				: BOOL;
		nServer1ErrorID				: UDINT;
END_VAR

IF bInit THEN 				// Init Step to close all sockets after login PLC with  downlaod
	fbSocketCloseAll(
		sSrvNetId:= '', 
		bExecute:= TRUE, 
		tTimeout:= T#3S, 
		bBusy=> , 
		bError=> bSocketCloseError, 
		nErrId=> nSocketCloseError);
	IF NOT (fbSocketCloseAll.bBusy OR fbSocketCloseAll.bError) THEN
		bInit := FALSE;
		fbSocketCloseAll(bExecute:= FALSE);
	END_IF
ELSE
		
	fbTcpEchoServer1(
		sLocalHost:= '127.0.0.1', 								// Server IP Adress
		nLocalPort:= nServer1Port, 									// Server port
		bStartCommunication:= bStartServer1Communication, 			// Allow Client-connection or close connection
		bConnected => bServer1Connected,							// Client connection is valid
		cmdData => cmdData,
		sSendData => sServerData,
		bBusy=> bServer1Busy, 
		bError=> bServer1Error, 
		nErrorID=> nServer1ErrorID);
END_IF

END_PROGRAM

// ---- VISUs/Main.TcVIS
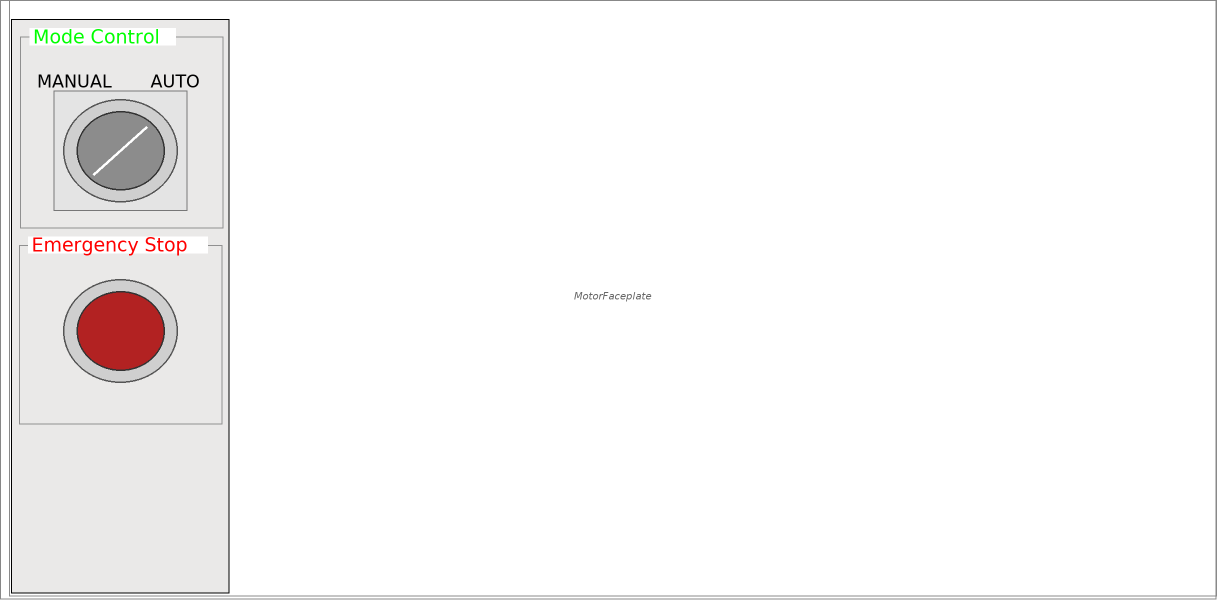
VISUALIZATION Main  // 1217x600
    TabControl (9,-4 1208x600)
        shows MotorFaceplate()
        shows MotorFaceplate2()
        [0]: TabTitle=Drive 1: Manual Control
        [1]: TabTitle=Drive 2
    Frame (11,19 218x574)
        shows SysPanel()
END_VISUALIZATION

// ---- VISUs/Templates/MotorFaceplate.TcVIS
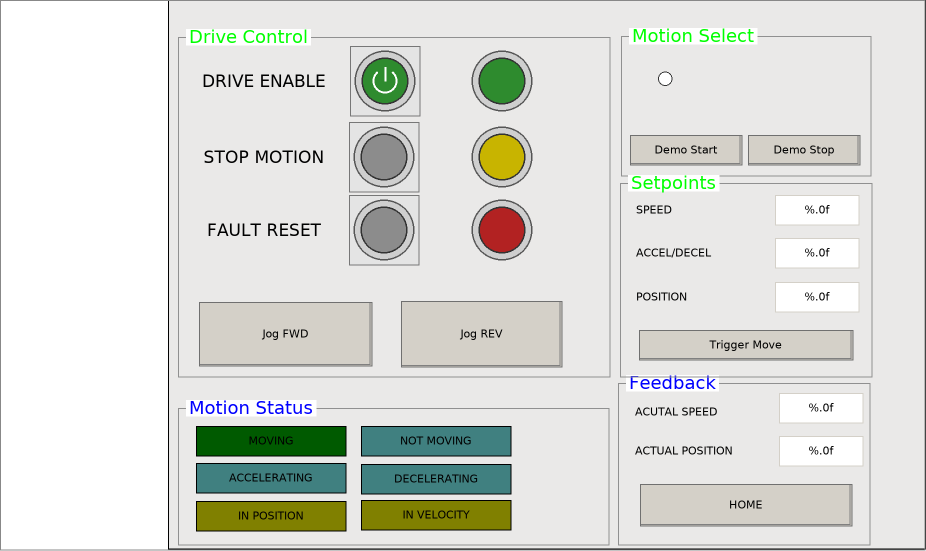
VISUALIZATION MotorFaceplate  // 926x551
    Rectangle (168,-2 758x551)
    GroupBox (178,29 432x348), "Drive Control"
        PowerSwitch (172,17 70x70), variable: ServoGVLs.servo1Interface.bDriveEnable, behaviour: TOGGLE, style: Switch-PowerSwitch-Green
        PushSwitch (171,93 70x70), variable: ServoGVLs.servo1Interface.bStopMotion, behaviour: TAP, style: Switch-PushSwitch-Gray
        PushSwitch (171,166 70x70), variable: ServoGVLs.servo1Interface.bFaultReset, behaviour: TAP, style: Switch-PushSwitch-Gray
        Lamp1 (289,17 70x70), variable: ServoGVLs.servo1Interface.bDriveEnabled, style: Lamp-Lamp1-Green
        Lamp1 (289,93 70x70), variable: ServoGVLs.servo1Interface.bNotMoving, style: Lamp-Lamp1-Yellow
        Lamp1 (289,166 70x70), variable: ServoGVLs.servo1Interface.bFaulted, style: Lamp-Lamp1-Red
        Label (11,37 150x30), "DRIVE ENABLE"
        Label (11,113 150x30), "STOP MOTION"
        Label (11,186 150x30), "FAULT RESET"
        Button (21,273 173x64), "Jog FWD"
            tap ServoGVLs.servo1Interface.bJogFWD
        Button (223,272 161x66), "Jog REV"
            tap ServoGVLs.servo1Interface.bJogRev
    GroupBox (178,400 431x145), "Motion Status"
        RoundedRectangle (18,26 150x30), "MOVING", colour toggle: ServoGVLs.servo1Interface.bMoving
        RoundedRectangle (183,26 150x30), "NOT MOVING", colour toggle: ServoGVLs.servo1Interface.bNotMoving
        RoundedRectangle (18,63 150x30), "ACCELERATING", colour toggle: ServoGVLs.servo1Interface.bAccelerating
        RoundedRectangle (183,64 150x30), "DECELERATING", colour toggle: ServoGVLs.servo1Interface.bDecelerating
        RoundedRectangle (18,101 150x30), "IN POSITION", colour toggle: ServoGVLs.servo1Interface.bInposition
        RoundedRectangle (183,100 150x30), "IN VELOCITY", colour toggle: ServoGVLs.servo1Interface.bInVelocity
    GroupBox (618,375 252x170), "Feedback"
        Textfield (161,18 84x30), "%.0f", text variable: ServoGVLs.servo1Interface.rActualSpeed
        Label (14,61 120x30), "ACTUAL POSITION"
        Textfield (161,61 84x30), "%.0f", text variable: ServoGVLs.servo1Interface.rActualPosition
        Label (14,22 108x30), "ACUTAL SPEED"
        Button (22,109 212x42), "HOME", invisible if: TRUE
            tap ServoGVLs.servo1Interface.bHome
    GroupBox (621,28 250x148), "Motion Select"
        RadioButton (35,21 173x59), variable: ServoGVLs.servo1Interface.iMotionSelect
            p3123465237: DEMO MODE
            p2481256679: RELATIVE POSITION
            p1032612214: VELOCITY CONTROL
        Button (9,107 112x30), "Demo Start", invisible if: ServoGVLs.servo1Interface.iMotionSelect = 0
            tap ServoGVLs.servo1Interface.bDemoModeStart
        Button (127,107 112x30), "Demo Stop", invisible if: ServoGVLs.servo1Interface.iMotionSelect = 0
            tap ServoGVLs.servo1Interface.bDemoModeStop
    GroupBox (620,175 252x202), "Setpoints"
        Label (13,20 76x30), "SPEED", invisible if: TRUE
        Textfield (155,20 84x30), "%.0f", text variable: ServoGVLs.servo1Interface.rSpeed, invisible if: TRUE
        Label (13,63 99x30), "ACCEL/DECEL", invisible if: TRUE
        Textfield (155,63 84x30), "%.0f", text variable: ServoGVLs.servo1Interface.rAccelDecel, invisible if: TRUE
        Label (13,107 76x30), "POSITION", invisible if: TRUE
        Textfield (155,107 84x30), "%.0f", text variable: ServoGVLs.servo1Interface.rPosition, invisible if: TRUE
        Button (19,155 214x30), "Trigger Move", invisible if: TRUE
            tap ServoGVLs.servo1Interface.bTriggerMove
END_VISUALIZATION

// ---- VISUs/Templates/MotorFaceplate2.TcVIS
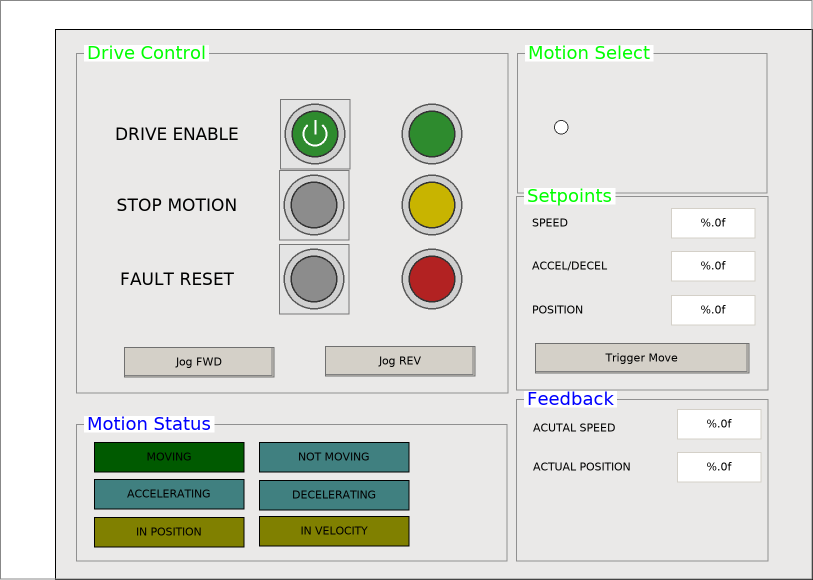
VISUALIZATION MotorFaceplate2  // 813x580
    Rectangle (55,29 758x551)
    GroupBox (76,45 432x348), "Drive Control"
        PowerSwitch (204,54 70x70), behaviour: TOGGLE, style: Switch-PowerSwitch-Green
        PushSwitch (203,125 70x70), behaviour: TOGGLE, style: Switch-PushSwitch-Gray
        PushSwitch (203,199 70x70), behaviour: TOGGLE, style: Switch-PushSwitch-Gray
        Lamp1 (321,54 70x70), style: Lamp-Lamp1-Green
        Lamp1 (321,125 70x70), style: Lamp-Lamp1-Yellow
        Lamp1 (321,199 70x70), style: Lamp-Lamp1-Red
        Label (26,74 150x30), "DRIVE ENABLE"
        Label (26,145 150x30), "STOP MOTION"
        Label (26,219 150x30), "FAULT RESET"
        Button (249,301 150x30), "Jog REV"
    GroupBox (517,45 250x148), "Motion Select"
        RadioButton (35,21 173x122), variable: ServoGVLs.servo1Interface.iMotionSelect
    GroupBox (516,188 252x202), "Setpoints"
        Label (13,20 76x30), "SPEED"
        Textfield (155,20 84x30), "%.0f"
        Label (13,63 99x30), "ACCEL/DECEL"
        Textfield (155,63 84x30), "%.0f"
        Label (13,107 76x30), "POSITION"
        Textfield (155,107 84x30), "%.0f"
        Button (19,155 214x30), "Trigger Move"
    GroupBox (76,416 431x145), "Motion Status"
        RoundedRectangle (18,26 150x30), "MOVING"
        RoundedRectangle (183,26 150x30), "NOT MOVING"
        RoundedRectangle (18,63 150x30), "ACCELERATING"
        RoundedRectangle (183,64 150x30), "DECELERATING"
        RoundedRectangle (18,101 150x30), "IN POSITION"
        RoundedRectangle (183,100 150x30), "IN VELOCITY"
    GroupBox (516,391 252x170), "Feedback"
        Textfield (161,18 84x30), "%.0f"
        Label (14,61 120x30), "ACTUAL POSITION"
        Textfield (161,61 84x30), "%.0f"
        Label (14,22 108x30), "ACUTAL SPEED"
    Button (124,347 150x30), "Jog FWD"
END_VISUALIZATION

// ---- VISUs/Templates/SysPanel.TcVIS
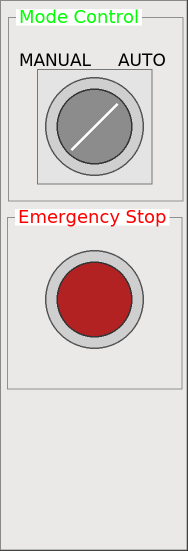
VISUALIZATION SysPanel  // 188x551
    Rectangle (0,0 188x551)
    GroupBox (8,9 175x192), "Mode Control"
        Label (4,36 86x30), "MANUAL"
        Label (105,36 58x30), "AUTO"
        RotarySwitch (29,60 115x115), variable: gvlMotion.manualMode, behaviour: TOGGLE, style: Switch-RotarySwitch-Gray
    GroupBox (7,209 175x180), "Emergency Stop"
        Lamp1 (30,33 115x115), tooltip "!", variable: TRUE, style: Lamp-Lamp1-Red
END_VISUALIZATION
